// Mitsubishi GX Works2 project: PLC Group1   PLC: FX3G

// global labels: Global1
VAR_GLOBAL
  Start_Day AT X007 : BOOL;
  Work_Day_Light AT Y000 : BOOL;
  Finish_Reset AT M8 : BOOL;
  Update_Stock AT M2 : BOOL;
  Check_Input AT M1 : BOOL;
  Output_Analog AT D8282 : INT;
  Input_Oat AT D2000 : REAL;
  Input_Helbon AT D2002 : REAL;
END_VAR
VAR_GLOBAL CONSTANT
  Helbon_For_Helbon : REAL := 320;
  Oat_For_Classic : REAL := 400;
END_VAR
VAR_GLOBAL
  Input_Honey AT D2004 : REAL;
END_VAR
VAR_GLOBAL CONSTANT
  Honey_For_Helbon : REAL := 160;
END_VAR
VAR_GLOBAL
  Stock_Oat AT D3000 : REAL;
  Stock_Helbon AT D3002 : REAL;
  Stock_Honey AT D3004 : REAL;
  Input_Analog1 AT D8280 : INT;
  Read_Input AT X003 : BOOL;
  Type_Snack AT D4200 : REAL;
END_VAR
VAR_GLOBAL CONSTANT
  Normalize : REAL := 403;
  Max_Regular : REAL := 5;
  Max_Classic : REAL := 5;
  Max_Helbon : REAL := 10;
  Min_Classic : REAL;
  Min_Helbon : REAL := 6;
END_VAR
VAR_GLOBAL
  Make_Classic AT M5 : BOOL;
  Make_Helbon AT M4 : BOOL;
  Check_Helbon AT M4 : BOOL;
  Check_Inventory AT M1 : BOOL;
  Mixer_On AT Y003 : BOOL;
END_VAR
VAR_GLOBAL CONSTANT
  Time_Mixing : WORD := 50;
END_VAR
VAR_GLOBAL
  Making_Time AT TC1 : BOOL;
  End_Making AT TS1 : BOOL;
  Inventory_Oat AT D2000 : REAL;
  Inventory_Helbon AT D2002 : REAL;
  Inventory_Honey AT D2004 : REAL;
END_VAR
VAR_GLOBAL CONSTANT
  Helbon_For_Classic : REAL := 160;
  Honey_For_Classic : REAL := 120;
END_VAR
VAR_GLOBAL
  Oven AT X002 : BOOL;
  Oven_On AT X002 : BOOL;
END_VAR
VAR_GLOBAL CONSTANT
  Blinking_Time : WORD := 5;
END_VAR
VAR_GLOBAL
  End_Blink6 AT TS6 : BOOL;
  End_Blink1 AT TS6 : BOOL;
  Blink1 AT TC6 : BOOL;
  Blink_Helper AT M7 : BOOL;
  Light1 AT Y001 : BOOL;
  End_Blink5 AT TS5 : BOOL;
  Mixing_Reg_Time AT TC3 : BOOL;
END_VAR
VAR_GLOBAL CONSTANT
  Mixing_Reg_Sec : WORD := 30;
END_VAR
VAR_GLOBAL
  Oven_Time_Helbon AT TC4 : BOOL;
  Oven_Time_Classic AT TC3 : BOOL;
END_VAR
VAR_GLOBAL CONSTANT
  Oven_Sec_Classic : WORD := 40;
END_VAR
VAR_GLOBAL
  End_Classic_Oven AT TS3 : BOOL;
  End_Helbon_Oven AT TS4 : BOOL;
  Light2 AT Y002 : BOOL;
  Ovenl_Time AT TC2 : BOOL;
END_VAR
VAR_GLOBAL CONSTANT
  Time_Oven_Sec : WORD := 80;
END_VAR
VAR_GLOBAL
  End_Oven AT TS2 : BOOL;
  Blink5 AT TC5 : BOOL;
  Start_Packing AT X006 : BOOL;
  Pack_One AT X000 : BOOL;
  First_Snack AT CC0 : BOOL;
END_VAR
VAR_GLOBAL CONSTANT
  Counter7 : WORD := 8;
  Counter8 : WORD := 8;
END_VAR
VAR_GLOBAL
  Counter_Pack AT CC1 : BOOL;
END_VAR
VAR_GLOBAL CONSTANT
  Counter1 : WORD := 1;
END_VAR
VAR_GLOBAL
  End_Counter1 AT CS0 : BOOL;
  End_Counter8 AT CS1 : BOOL;
  Light4 AT Y004 : BOOL;
  Packs_Amount AT D5000 : REAL;
END_VAR
VAR_GLOBAL CONSTANT
  Add_One : REAL := 1;
END_VAR
VAR_GLOBAL
  End_Day AT M0 : BOOL;
  Emergency_Stop AT X005 : BOOL;
END_VAR
VAR_GLOBAL CONSTANT
  Normalize_Back : REAL := 40.45;
END_VAR
VAR_GLOBAL
  Oat_Oven AT D4204 : REAL;
  Oat_Heating AT D4204 : REAL;
  Mixing_Classic AT D4202 : REAL;
END_VAR
VAR_GLOBAL CONSTANT
  Total_Classic : REAL := 680;
  Total_Helbon : REAL := 720;
END_VAR
VAR_GLOBAL
  Mixing_Helbon AT D4204 : REAL;
  Baking_Bowl AT D4206 : REAL;
  Down54 AT M9 : BOOL;
  Indicator AT M9 : BOOL;
  Continue AT M70 : BOOL;
  Check_stock AT M69 : BOOL;
END_VAR
VAR_GLOBAL CONSTANT
  zero_oat : REAL;
  zero_helbon : REAL;
  zero_honey : REAL;
END_VAR
VAR_GLOBAL
  Reset45 AT M18 : BOOL;
  Fiktivit AT M88 : BOOL;
  Indicator_Stock AT M99 : BOOL;
  CheckCheck AT M44 : BOOL;
END_VAR

// task Task_01 (event TRUE, interval 0, priority 31): POU_01

PROGRAM POU_01
VAR CONSTANT
  Oat_For_Helbon : REAL := 160;
  Oven_Sec_Helbon : WORD := 50;
END_VAR
VAR
  Check54 : BOOL;
END_VAR
(* structured ladder/FBD written out as ST: instructions are called as NAME(EN, inputs, outputs); _pN, _eN, _tN stand for wires *)
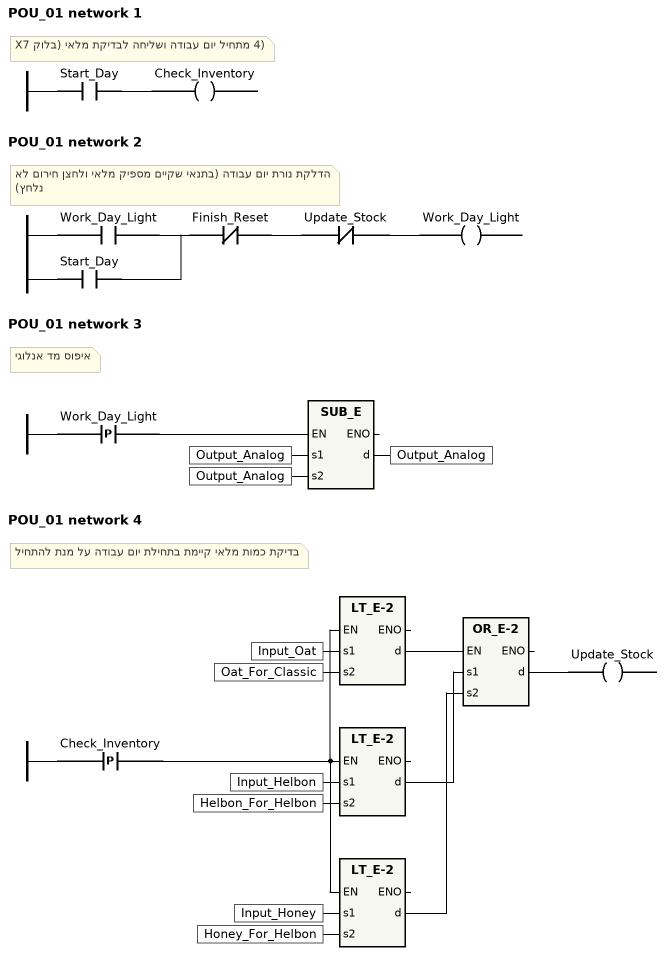
(* network 1 *)
(* X7 מתחיל יום עבודה ושליחה לבדיקת מלאי (בלוק 4) *)
Check_Inventory := Start_Day;
(* network 2 *)
(* הדלקת נורת יום עבודה (בתנאי שקיים מספיק מלאי ולחצן חירום לא נלחץ) *)
Work_Day_Light := ((Work_Day_Light OR Start_Day) AND NOT Finish_Reset) AND NOT Update_Stock;
(* network 3 *)
(* איפוס מד אנלוגי *)
SUB_E(LDP(TRUE, Work_Day_Light), Output_Analog, Output_Analog, Output_Analog);
(* network 4 *)
(* בדיקת כמות מלאי קיימת בתחילת יום עבודה על מנת להתחיל *)
_p1 := LDP(TRUE, Check_Inventory);
LT_E(_p1, Input_Oat, Oat_For_Classic, _t2);
LT_E(_p1, Input_Helbon, Helbon_For_Helbon, _t3);
LT_E(_p1, Input_Honey, Honey_For_Helbon, _t4);
OR_E(_t2, _t3, _t4, _t5);
Update_Stock := _t5;
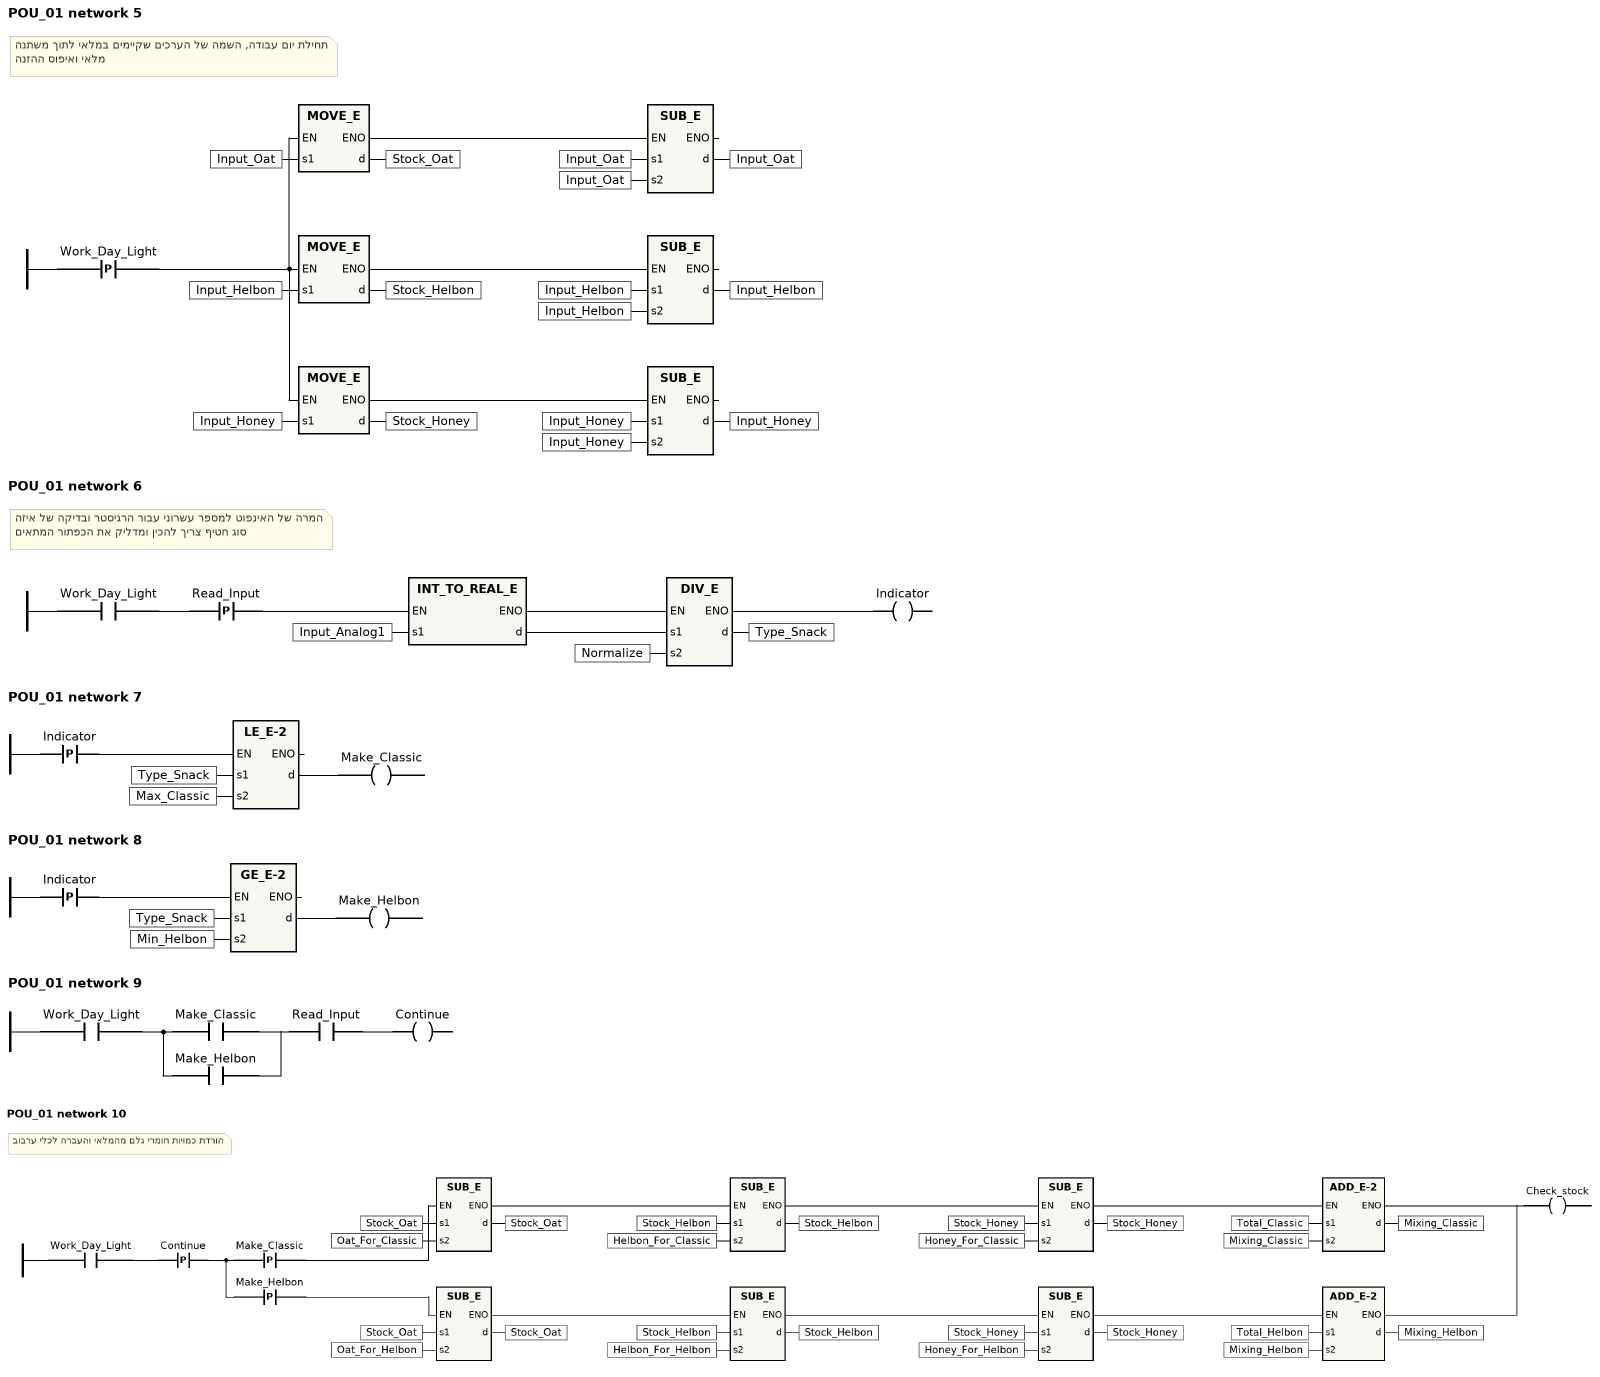
(* network 5 *)
(* תחילת יום עבודה, השמה של הערכים שקיימים במלאי לתוך משתנה מלאי ואיפוס ההזנה *)
_p1 := LDP(TRUE, Work_Day_Light);
_e2 := MOVE_E(_p1, Input_Oat, Stock_Oat);
SUB_E(_e2, Input_Oat, Input_Oat, Input_Oat);
_e3 := MOVE_E(_p1, Input_Helbon, Stock_Helbon);
SUB_E(_e3, Input_Helbon, Input_Helbon, Input_Helbon);
_e4 := MOVE_E(_p1, Input_Honey, Stock_Honey);
SUB_E(_e4, Input_Honey, Input_Honey, Input_Honey);
(* network 6 *)
(* המרה של האינפוט למספר עשרוני עבור הרגיסטר ובדיקה של איזה סוג חטיף צריך להכין ומדליק את הכפתור המתאים *)
_e2 := INT_TO_REAL_E(Work_Day_Light AND LDP(TRUE, Read_Input), Input_Analog1, _t1);
_e3 := DIV_E(_e2, _t1, Normalize, Type_Snack);
Indicator := _e3;
(* network 7 *)
LE_E(LDP(TRUE, Indicator), Type_Snack, Max_Classic, _t1);
Make_Classic := _t1;
(* network 8 *)
GE_E(LDP(TRUE, Indicator), Type_Snack, Min_Helbon, _t1);
Make_Helbon := _t1;
(* network 9 *)
Continue := ((Work_Day_Light AND Make_Classic) OR (Work_Day_Light AND Make_Helbon)) AND Read_Input;
(* network 10 *)
(* הורדת כמויות חומרי גלם מהמלאי והעברה לכלי ערבוב *)
_p1 := Work_Day_Light AND LDP(TRUE, Continue);
_e2 := SUB_E(_p1 AND LDP(TRUE, Make_Classic), Stock_Oat, Oat_For_Classic, Stock_Oat);
_e3 := SUB_E(_e2, Stock_Helbon, Helbon_For_Classic, Stock_Helbon);
_e4 := SUB_E(_e3, Stock_Honey, Honey_For_Classic, Stock_Honey);
_e5 := ADD_E(_e4, Total_Classic, Mixing_Classic, Mixing_Classic);
_e6 := SUB_E(_p1 AND LDP(TRUE, Make_Helbon), Stock_Oat, Oat_For_Helbon, Stock_Oat);
_e7 := SUB_E(_e6, Stock_Helbon, Helbon_For_Helbon, Stock_Helbon);
_e8 := SUB_E(_e7, Stock_Honey, Honey_For_Helbon, Stock_Honey);
_e9 := ADD_E(_e8, Total_Helbon, Mixing_Helbon, Mixing_Helbon);
Check_stock := _e5 OR _e9;
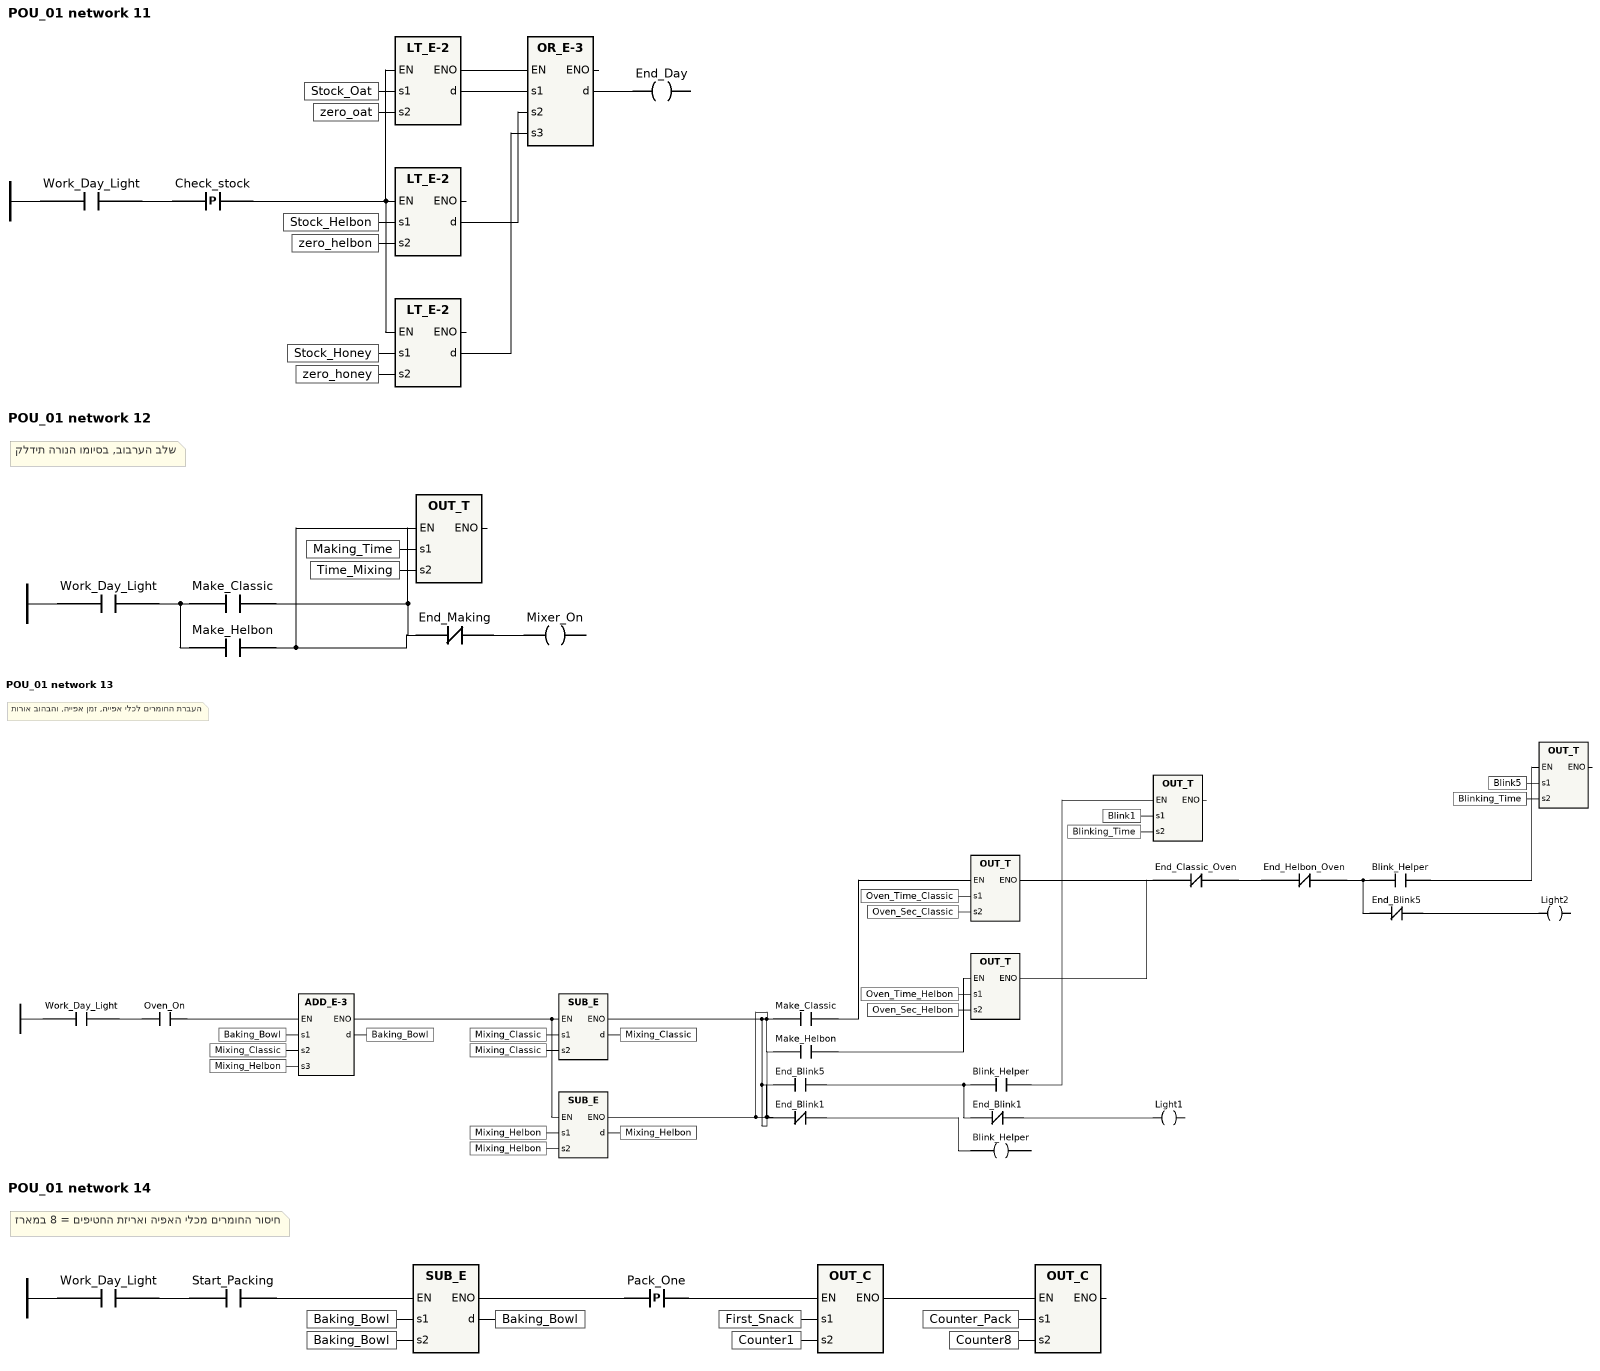
(* network 11 *)
_p1 := Work_Day_Light AND LDP(TRUE, Check_stock);
_e3 := LT_E(_p1, Stock_Oat, zero_oat, _t2);
LT_E(_p1, Stock_Helbon, zero_helbon, _t4);
LT_E(_p1, Stock_Honey, zero_honey, _t5);
OR_E(_e3, _t2, _t4, _t5, _t6);
End_Day := _t6;
(* network 12 *)
(* שלב הערבוב, בסיומו הנורה תידלק *)
_p1 := (Work_Day_Light AND Make_Classic) OR (Work_Day_Light AND Make_Helbon);
OUT_T(_p1, Making_Time, Time_Mixing);
Mixer_On := _p1 AND NOT End_Making;
(* network 13 *)
(* העברת החומרים לכלי אפייה, זמן אפייה, והבהוב אורות *)
_e1 := ADD_E(Work_Day_Light AND Oven_On, Baking_Bowl, Mixing_Classic, Mixing_Helbon, Baking_Bowl);
_e2 := SUB_E(_e1, Mixing_Classic, Mixing_Classic, Mixing_Classic);
_e3 := SUB_E(_e1, Mixing_Helbon, Mixing_Helbon, Mixing_Helbon);
_p4 := _e2 OR _e3;
_e5 := OUT_T(_p4 AND Make_Classic, Oven_Time_Classic, Oven_Sec_Classic);
_e6 := OUT_T(_p4 AND Make_Helbon, Oven_Time_Helbon, Oven_Sec_Helbon);
_p7 := ((_e5 OR _e6) AND NOT End_Classic_Oven) AND NOT End_Helbon_Oven;
OUT_T(_p7 AND Blink_Helper, Blink5, Blinking_Time);
Light2 := _p7 AND NOT End_Blink5;
_p8 := _p4 AND End_Blink5;
OUT_T(_p8 AND Blink_Helper, Blink1, Blinking_Time);
Light1 := _p8 AND NOT End_Blink1;
Blink_Helper := _p4 AND NOT End_Blink1;
(* network 14 *)
(* חיסור החומרים מכלי האפיה ואריזת החטיפים = 8 במארז *)
_e1 := SUB_E(Work_Day_Light AND Start_Packing, Baking_Bowl, Baking_Bowl, Baking_Bowl);
_e2 := OUT_C(_e1 AND LDP(TRUE, Pack_One), First_Snack, Counter1);
OUT_C(_e2, Counter_Pack, Counter8);
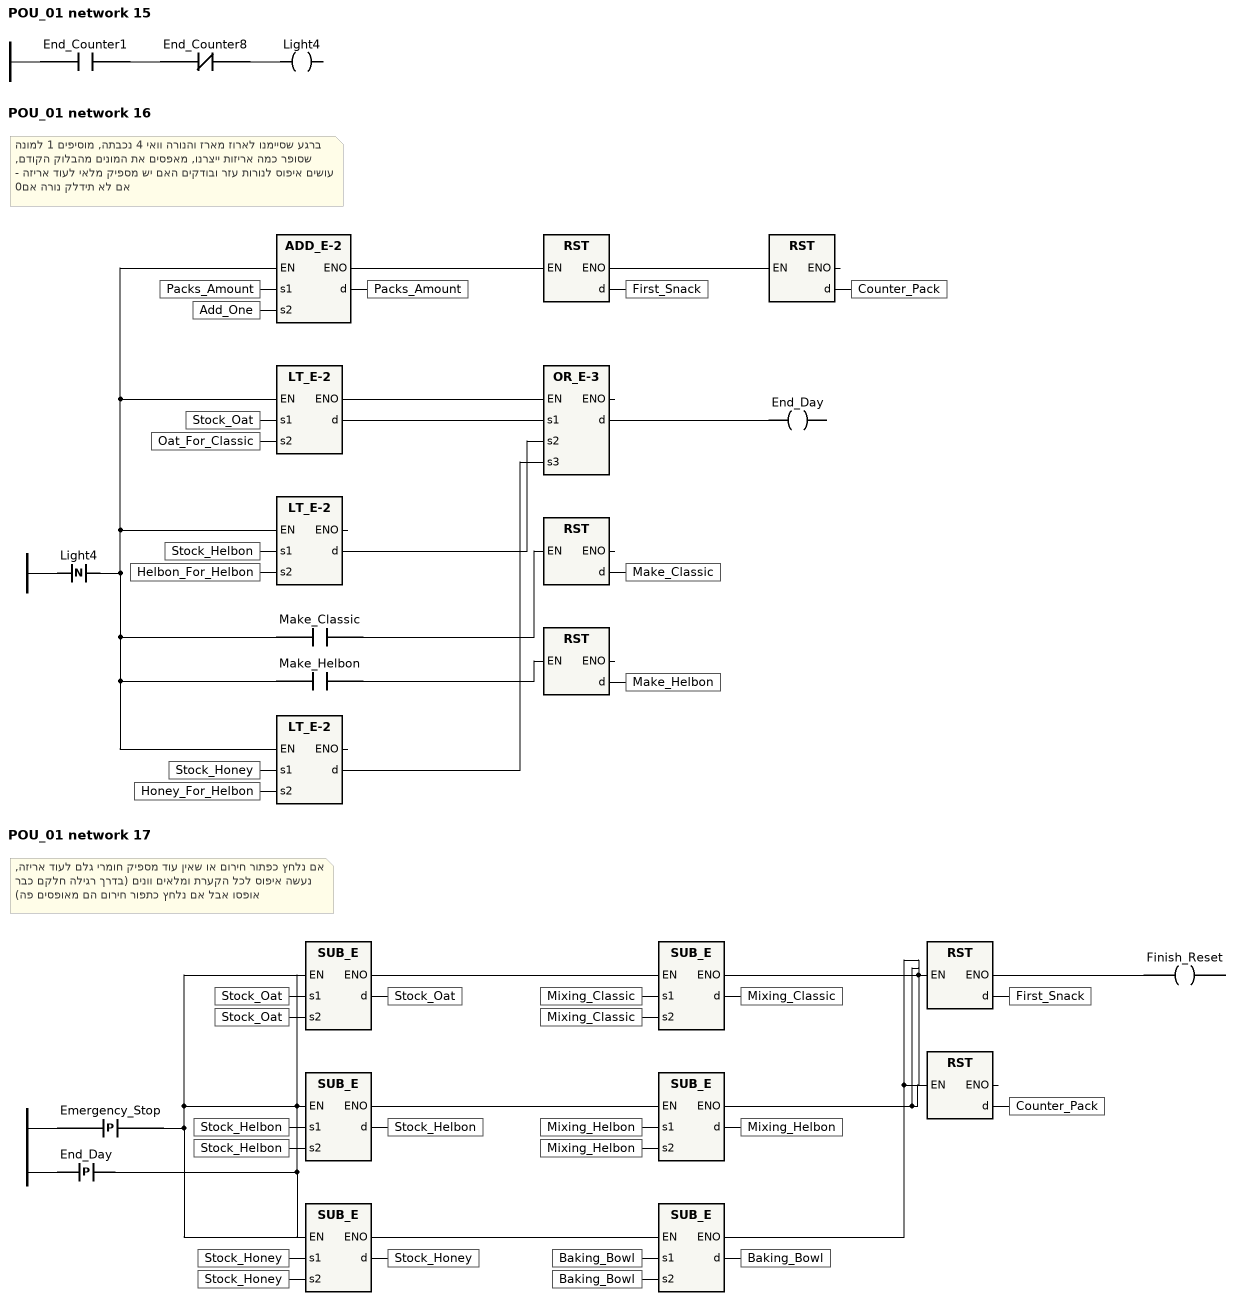
(* network 15 *)
Light4 := End_Counter1 AND NOT End_Counter8;
(* network 16 *)
(* ברגע שסיימנו לארוז מארז והנורה וואי 4 נכבתה, מוסיפים 1 למונה שסופר כמה אריזות ייצרנו, מאפסים את המונים מהבלוק הקודם, עושים איפוס לנורות עזר ובודקים האם יש מספיק מלאי לעוד אריזה - אם לא תידלק נורה אם0 *)
_p1 := LDF(TRUE, Light4);
_e2 := ADD_E(_p1, Packs_Amount, Add_One, Packs_Amount);
_e3 := RST(_e2, First_Snack);
RST(_e3, Counter_Pack);
_e5 := LT_E(_p1, Stock_Oat, Oat_For_Classic, _t4);
RST(_p1 AND Make_Classic, Make_Classic);
RST(_p1 AND Make_Helbon, Make_Helbon);
LT_E(_p1, Stock_Helbon, Helbon_For_Helbon, _t6);
LT_E(_p1, Stock_Honey, Honey_For_Helbon, _t7);
OR_E(_e5, _t4, _t6, _t7, _t8);
End_Day := _t8;
(* network 17 *)
(* אם נלחץ כפתור חירום או שאין עוד מספיק חומרי גלם לעוד אריזה, נעשה איפוס לכל הקערת ומלאים וונים (בדרך רגילה חלקם כבר אופסו אבל אם נלחץ כתפור חירום הם מאופסים פה) *)
_p1 := LDP(TRUE, Emergency_Stop) OR LDP(TRUE, End_Day);
_e2 := SUB_E(_p1, Stock_Oat, Stock_Oat, Stock_Oat);
_e3 := SUB_E(_e2, Mixing_Classic, Mixing_Classic, Mixing_Classic);
_e4 := SUB_E(_p1, Stock_Helbon, Stock_Helbon, Stock_Helbon);
_e5 := SUB_E(_e4, Mixing_Helbon, Mixing_Helbon, Mixing_Helbon);
_e6 := SUB_E(_p1, Stock_Honey, Stock_Honey, Stock_Honey);
_e7 := SUB_E(_e6, Baking_Bowl, Baking_Bowl, Baking_Bowl);
_p8 := _e3 OR _e5 OR _e7;
_e9 := RST(_p8, First_Snack);
Finish_Reset := _e9;
RST(_p8, Counter_Pack);
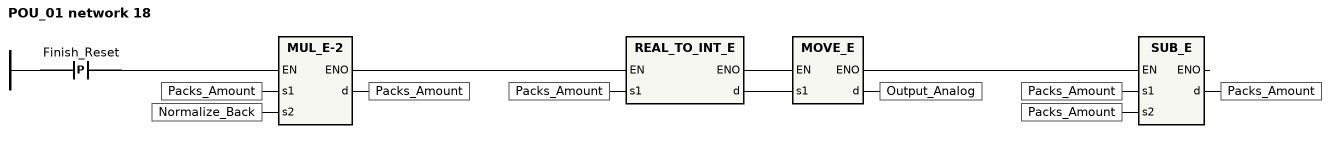
(* network 18 *)
_e1 := MUL_E(LDP(TRUE, Finish_Reset), Packs_Amount, Normalize_Back, Packs_Amount);
_e3 := REAL_TO_INT_E(_e1, Packs_Amount, _t2);
_e4 := MOVE_E(_e3, _t2, Output_Analog);
SUB_E(_e4, Packs_Amount, Packs_Amount, Packs_Amount);
END_PROGRAM
